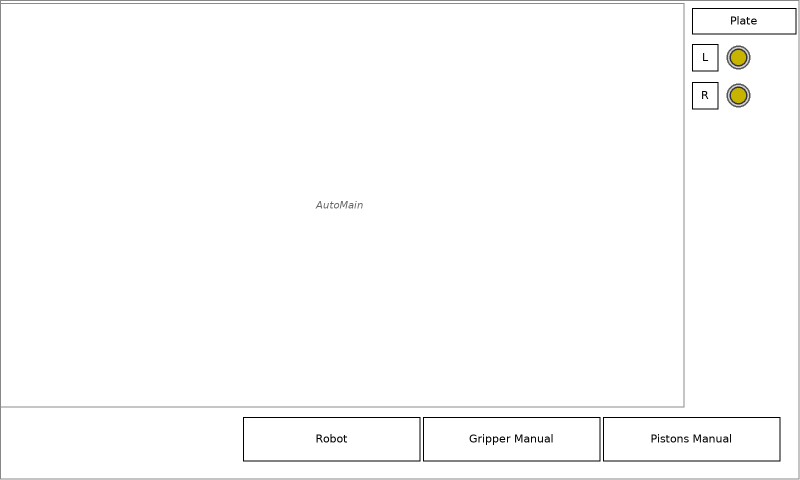
VISUALIZATION Main  // 800x480
    Rectangle (603,417 177x44), "Pistons Manual"
        OnMouseDown: change screen: PistonsManual
    Rectangle (243,417 177x44), "Robot"
        OnMouseDown: change screen: Robot
    Rectangle (423,417 177x44), "Gripper Manual"
        OnMouseDown: change screen: GripperManual
    Frame (-4,3 688x404)
        shows AutoMain(stMasterAutoCycle := GVL_HMI.stMasterAuto, stCfg := GVL_HmiPersistent.stMasterAutoCfg)
    Rectangle (692,8 104x26), "Plate"
    Rectangle (692,44 26x27), "L"
    Lamp1 (724,44 29x27), variable: GVL_HMI.bPlateSenL, style: Lamp-Lamp1-Yellow
    Rectangle (692,82 26x27), "R"
    Lamp1 (724,82 29x27), variable: GVL_HMI.bPlateSenR, style: Lamp-Lamp1-Yellow
END_VISUALIZATION

(* stored: Version 1.1.0.1, ProductVersion 3.1.4024.16
   Visu Main: Id {7fac2d1c-350f-4a9f-ac48-46c0699392e3} *)
